// TIA Portal V19 export
DATA_BLOCK "MODBUS DB"   // DB53
{ S7_Optimized_Access := 'FALSE' }
   VAR
      "STEP" : Int;
      EDGE : Bool;
      P_TRIG : Struct
         "0" : Bool;
         "1" : Bool;
         "2" : Bool;
         "3" : Bool;
         "4" : Bool;
         "5" : Bool;
         "6" : Bool;
         "7" : Bool;
         "8" : Bool;
         "9" : Bool;
         "10" : Bool;
         "11" : Bool;
         "12" : Bool;
         "13" : Bool;
         "14" : Bool;
         "15" : Bool;
         "16" : Bool;
         "17" : Bool;
         "18" : Bool;
         "19" : Bool;
         "20" : Bool;
         "21" : Bool;
         "22" : Bool;
         "23" : Bool;
         "24" : Bool;
         "25" : Bool;
         "26" : Bool;
         "27" : Bool;
         "28" : Bool;
         "29" : Bool;
         "30" : Bool;
         "31" : Bool;
         "32" : Bool;
         "33" : Bool;
         "34" : Bool;
         "35" : Bool;
         "36" : Bool;
         "37" : Bool;
         "38" : Bool;
         "39" : Bool;
         "40" : Bool;
         "41" : Bool;
         "42" : Bool;
         "43" : Bool;
         "44" : Bool;
         "45" : Bool;
         "46" : Bool;
         "47" : Bool;
         "48" : Bool;
         "49" : Bool;
         "50" : Bool;
      END_STRUCT;
      VFD_1 : Struct
         WRITE : Struct
            DONE : Bool;
            BUSY : Bool;
            ERROR : Bool;
            STATUS : Int;
         END_STRUCT;
         READ : Struct
            DONE : Bool;
            BUSY : Bool;
            ERROR : Bool;
            STATUS : Int;
         END_STRUCT;
      END_STRUCT;
      "VFD_1 SEND" : UInt;
      "VFD_1 RECEIVE" : UInt;
      VFD_2 : Struct
         WRITE : Struct
            DONE : Bool;
            BUSY : Bool;
            ERROR : Bool;
            STATUS : Int;
         END_STRUCT;
         READ : Struct
            DONE : Bool;
            BUSY : Bool;
            ERROR : Bool;
            STATUS : Int;
         END_STRUCT;
      END_STRUCT;
      "VFD_2 SEND" : UInt;
      "VFD_2 RECEIVE" : UInt;
      VFD_3 : Struct
         WRITE : Struct
            DONE : Bool;
            BUSY : Bool;
            ERROR : Bool;
            STATUS : Int;
         END_STRUCT;
         READ : Struct
            DONE : Bool;
            BUSY : Bool;
            ERROR : Bool;
            STATUS : Int;
         END_STRUCT;
      END_STRUCT;
      "VFD_3 SEND" : UInt;
      "VFD_3 RECEIVE" : UInt;
      VFD_4 : Struct
         WRITE : Struct
            DONE : Bool;
            BUSY : Bool;
            ERROR : Bool;
            STATUS : Int;
         END_STRUCT;
         READ : Struct
            DONE : Bool;
            BUSY : Bool;
            ERROR : Bool;
            STATUS : Int;
         END_STRUCT;
      END_STRUCT;
      "VFD_4 SEND" : UInt;
      "VFD_4 RECEIVE" : UInt;
      VFD_5 : Struct
         WRITE : Struct
            DONE : Bool;
            BUSY : Bool;
            ERROR : Bool;
            STATUS : Int;
         END_STRUCT;
         READ : Struct
            DONE : Bool;
            BUSY : Bool;
            ERROR : Bool;
            STATUS : Int;
         END_STRUCT;
      END_STRUCT;
      "VFD_5 SEND" : UInt;
      "VFD_5 RECEIVE" : UInt;
      VFD_6 : Struct
         WRITE : Struct
            DONE : Bool;
            BUSY : Bool;
            ERROR : Bool;
            STATUS : Int;
         END_STRUCT;
         READ : Struct
            DONE : Bool;
            BUSY : Bool;
            ERROR : Bool;
            STATUS : Int;
         END_STRUCT;
      END_STRUCT;
      "VFD_6 SEND" : UInt;
      "VFD_6 RECEIVE" : UInt;
      VFD_7 : Struct
         WRITE : Struct
            DONE : Bool;
            BUSY : Bool;
            ERROR : Bool;
            STATUS : Int;
         END_STRUCT;
         READ : Struct
            DONE : Bool;
            BUSY : Bool;
            ERROR : Bool;
            STATUS : Int;
         END_STRUCT;
      END_STRUCT;
      "VFD_7 SEND" : UInt;
      "VFD_7 RECEIVE" : UInt;
   END_VAR
BEGIN
END_DATA_BLOCK
